TYPE CmpConvStop : //Version 03 - 06/17/2022
STRUCT
	
	Framework: Framework;
	Available: BOOL;
	Release: BOOL;
	WorkReq: BOOL;
	WorkCmp: BOOL;
	ConvRunning: BOOL;
	StatusInCycleAuto: BOOL;
	StatusPuckPresent: BOOL;
	StatusBufferFull: BOOL;
	RemoteBufferFull: BOOL;
	FreeRunCycleStop: BOOL;
	Config: CmpConvStopConfig;
	
END_STRUCT
END_TYPE

(* stored: Version 1.1.0.1, ProductVersion 3.1.4024.6
   DUT CmpConvStop: Id {1bd4892d-4f24-498a-82b8-a1d7b14138da} *)
